// TIA Portal V20 export
VAR_GLOBAL   // PLC tag table "Conveyor 1"
   B_lightBarrier_C1 AT %I104.0 : Bool;   // Lichtschranke / Light barrier
   S_bay1_C1 AT %I104.1 : Bool;   // Taster Platz 1 / Momentary contact Bay 1
   S_bay2_C1 AT %I104.2 : Bool;   // Taster Platz 2 / Momentary contact Bay 2
   S_bay3_C1 AT %I104.3 : Bool;   // Taster Platz 3 / Momentary contact Bay 3
   S_lightBarrier_C1 AT %I104.4 : Bool;   // Taster Lichtschranken-Platz / Momentary contact Light barrier bay
   B_bay1_C1 AT %I104.5 : Bool;   // Initiator Platz 1 / Proximity sensor Bay 1
   B_bay2_C1 AT %I104.6 : Bool;   // Initiator Platz 2 / Proximity sensor Bay 2
   B_bay3_C1 AT %I104.7 : Bool;   // Initiator Platz 3 / Proximity sensor Bay 3
   P_bay1_C1 AT %Q104.1 : Bool;   // Meldeleuchte Platz 1 / Indicator light Bay 1
   P_bay2_C1 AT %Q104.2 : Bool;   // Meldeleuchte Platz 2 / Indicator light Bay 2
   P_bay3_C1 AT %Q104.3 : Bool;   // Meldeleuchte Platz 3 / Indicator light Bay 3
   P_lightBarrier_C1 AT %Q104.4 : Bool;   // Meldeleuchte Lichtschranken-Platz / Indicator light Light barrier bay
   K_right_C1 AT %Q104.5 : Bool;   // Bandmotor Rechts / Run conveyor RIGHT
   K_left_C1 AT %Q104.6 : Bool;   // Bandmotor Links / Run conveyor LEFT
   P_horn_C1 AT %Q104.7 : Bool;   // Hupe / Horn
   S_slider2_C1 AT %IW130 : Int;   // Slider 2
   P_ao1_C1 AT %QW130 : Int;   // Analog output 1
   P_display1_C1 AT %QW132 : Int;   // Analog display 1
   P_display2_C1 AT %QW134 : Int;   // Analog display 2
END_VAR
